Fanuc KAREL source: kc00009.KL

PROGRAM KC00009
%STACKSIZE=65535
%PRIORITY=65535
%NOLOCKGROUP
VAR
I : INTEGER
J : INTEGER
K : INTEGER
R : REAL
B : BOOLEAN
S : STRING[80]
T : STRING[80]
AI : ARRAY[8] OF INTEGER
AB : ARRAY[244] OF BYTE
-- UNRESOLVED DECLARATIONS (source type spelling not recovered)
-- P : TYPE_0x001F (type_u16=0x001F)
-- Q : TYPE_0x001F (type_u16=0x001F)
BEGIN
INSERT_NODE(P,I,J)
END KC00009
